# B&R Automation Studio project A2019059_Linka_Power_CP (part 4)

### Hardware.hwl.2.mine
```
BR.AS.HardwareTopology (Version=0.0.0.1)
  TimeStamps:
    TimeStamp (LogicalPath=Config1.Hardware.hw, LastWriteTime=07/08/2020 07:45:30)
  Modules:
    Module PC1 (Type=5PC910.SX02-00, X=2263, Y=-320)
    Module 5AC901.IUPS-01 (Type=5AC901.IUPS-01, X=2322, Y=-217)
    Module 5AC901.BX02-00 (Type=5AC901.BX02-00, X=2322, Y=-287)
    Module 5ACPCI_XPNM_00 (Type=5ACPCI.XPNM-00, X=2327, Y=-245)
    Module 5LS182.6-1 (Type=5LS182.6-1, X=2327, Y=-274)
    Module 5PC900_TS17_00 (Type=5PC900.TS17-00, X=2322, Y=-310)
    Module AB1.0 (Type=6PPT50.156B-10B, X=-440, Y=-300)
    Module AB2.0 (Type=6PPT50.156B-10B, X=672, Y=-281)
    Module AB4.0 (Type=6PPT50.156B-10B, X=3220, Y=-302)
    Module 0AC808.9-1 (Type=0AC808.9-1, X=2483, Y=-229)
    Module X20BB81 (Type=X20BB81, X=-440, Y=20)
    Module X20BM33 (Type=X20BM33, X=-377, Y=20)
    Module AB1.4_20xSI (Type=X20SI9100, X=-377, Y=20)
    Module X20TB52b (Type=X20TB52, X=-364, Y=46)
    Module X20TB52a (Type=X20TB52, X=-377, Y=46)
    Module X20BM33d (Type=X20BM33, X=-351, Y=20)
    Module AB1.5_6xSO (Type=X20SO6530, X=-351, Y=20)
    Module X20TB72 (Type=X20TB72, X=-351, Y=46)
    Module X20BM11 (Type=X20BM11, X=-325, Y=20)
    Module AB1.6_16xDI (Type=X20DIF371, X=-325, Y=20)
    Module X20TB1F (Type=X20TB1F, X=-325, Y=47)
    Module X20BM11a (Type=X20BM11, X=-312, Y=20)
    Module AB1.7_16xDI (Type=X20DIF371, X=-312, Y=20)
    Module X20TB1F1 (Type=X20TB1F, X=-312, Y=47)
    Module X20BM11b (Type=X20BM11, X=-299, Y=20)
    Module AB1.8_16xDO (Type=X20DOF322, X=-299, Y=20)
    Module X20TB1F2 (Type=X20TB1F, X=-299, Y=47)
    Module X20BM11c (Type=X20BM11, X=-286, Y=20)
    Module AB1.9_16xDO (Type=X20DOF322, X=-286, Y=20)
    Module X20TB1F3 (Type=X20TB1F, X=-286, Y=47)
    Module X20BM11h (Type=X20BM11, X=-273, Y=20)
    Module AB1.10_X2X (Type=X20BT9400, X=-273, Y=20)
    Module X20TB12d (Type=X20TB12, X=-273, Y=47)
    Module AB1.3_Napajanie (Type=X20PS9400, X=-390, Y=20)
    Module X20TB12 (Type=X20TB12, X=-390, Y=47)
    Module AB1.2_Powerlink (Type=X20BC1083, X=-415, Y=20)
    Module X20BB81a (Type=X20BB81, X=720, Y=20)
    Module X20BM33a (Type=X20BM33, X=783, Y=20)
    Module AB2.4_20xSI (Type=X20SI9100, X=783, Y=20)
    Module X20TB52d (Type=X20TB52, X=796, Y=46)
    Module X20TB52c (Type=X20TB52, X=783, Y=46)
    Module X20BM33e (Type=X20BM33, X=809, Y=20)
    Module AB2.5_6xSO (Type=X20SO6530, X=809, Y=20)
    Module X20TB72a (Type=X20TB72, X=809, Y=46)
    Module X20BM33h (Type=X20BM33, X=835, Y=20)
    Module AB2.6_6xSO (Type=X20SO6530, X=835, Y=20)
    Module X20TB72d (Type=X20TB72, X=835, Y=46)
    Module X20BM11d (Type=X20BM11, X=861, Y=20)
    Module AB2.7_16xDI (Type=X20DIF371, X=861, Y=20)
    Module X20TB1F4 (Type=X20TB1F, X=861, Y=47)
    Module X20BM11e (Type=X20BM11, X=874, Y=20)
    Module AB2.8_16xDI (Type=X20DIF371, X=874, Y=20)
    Module X20TB1F5 (Type=X20TB1F, X=874, Y=47)
    Module X20BM11l (Type=X20BM11, X=887, Y=20)
    Module AB2.9_16xDO (Type=X20DOF322, X=887, Y=20)
    Module X20TB1F8 (Type=X20TB1F, X=887, Y=47)
    Module X20BM11m (Type=X20BM11, X=900, Y=20)
    Module AB2.10_16xDO (Type=X20DOF322, X=900, Y=20)
    Module X20TB1F9 (Type=X20TB1F, X=900, Y=47)
    Module X20BM11i (Type=X20BM11, X=913, Y=20)
    Module AB2.11_X2X (Type=X20BT9400, X=913, Y=20)
    Module X20TB12e (Type=X20TB12, X=913, Y=47)
    Module AB2.3_Napajanie (Type=X20PS9400, X=770, Y=20)
    Module X20TB12a (Type=X20TB12, X=770, Y=47)
    Module AB2.2_Powerlink (Type=X20BC1083, X=745, Y=20)
    Module X20BB81b (Type=X20BB81, X=2019, Y=20)
    Module X20BM11f (Type=X20BM11, X=2082, Y=20)
    Module AB3.7_16xDI (Type=X20DIF371, X=2082, Y=20)
    Module X20TB1F6 (Type=X20TB1F, X=2082, Y=47)
    Module X20BM11g (Type=X20BM11, X=2095, Y=20)
    Module AB3.8_16xDO (Type=X20DOF322, X=2095, Y=20)
    Module X20TB1F7 (Type=X20TB1F, X=2095, Y=47)
    Module X20BM33b (Type=X20BM33, X=2108, Y=20)
    Module AB3.5_20xSI (Type=X20SI9100, X=2108, Y=20)
    Module X20TB52f (Type=X20TB52, X=2121, Y=46)
    Module X20TB52e (Type=X20TB52, X=2108, Y=46)
    Module X20BM33f (Type=X20BM33, X=2134, Y=20)
    Module AB3.6_6xSO (Type=X20SO6530, X=2134, Y=20)
    Module X20TB72b (Type=X20TB72, X=2134, Y=46)
    Module X20BM11j (Type=X20BM11, X=2160, Y=20)
    Module AB3.9_X2X (Type=X20BT9400, X=2160, Y=20)
    Module X20TB12f (Type=X20TB12, X=2160, Y=47)
    Module AB3.3_Napajanie (Type=X20PS9400, X=2069, Y=20)
    Module X20TB12b (Type=X20TB12, X=2069, Y=47)
    Module AB3.2_Powerlink (Type=X20BC1083, X=2044, Y=20)
    Module X20BB81c (Type=X20BB81, X=3240, Y=-2)
    Module X20BM33c (Type=X20BM33, X=3303, Y=-2)
    Module SI4.0 (Type=X20SI9100, X=3303, Y=-2)
    Module X20TB52h (Type=X20TB52, X=3316, Y=24)
    Module X20TB52g (Type=X20TB52, X=3303, Y=24)
    Module X20BM33g (Type=X20BM33, X=3329, Y=-2)
    Module SO4.0 (Type=X20SO6530, X=3329, Y=-2)
    Module X20TB72c (Type=X20TB72, X=3329, Y=24)
    Module X20BM11k (Type=X20BM11, X=3355, Y=-2)
    Module BT4.0 (Type=X20BT9400, X=3355, Y=-2)
    Module X20TB12g (Type=X20TB12, X=3355, Y=25)
    Module PS4.0 (Type=X20PS9400, X=3290, Y=-2)
    Module X20TB12c (Type=X20TB12, X=3290, Y=25)
    Module BC4.0 (Type=X20BC1083, X=3265, Y=-2)
    Module SL1_SafetyMaster (Type=X20SL8100, X=2283, Y=20)
    Module X20TB52 (Type=X20TB52, X=2330, Y=47)
    Module X20MK0211 (Type=X20MK0211, X=2286, Y=90)
    Module DM4.0 (Type=X67DM1321.L12, X=3210, Y=523)
    Module DM3.1 (Type=X67DM1321.L12, X=2090, Y=525)
    Module DM2.1_16DI/DO (Type=X67DM1321.L12, X=1024, Y=525)
    Module DM1.1_16DI/DO (Type=X67DM1321.L12, X=-282, Y=525)
    Module SI1.1 (Type=X67SI8103, X=-364, Y=525)
    Module SI1.2 (Type=X67SI8103, X=146, Y=525)
    Module SI2.1 (Type=X67SI8103, X=815, Y=525)
    Module SI2.2 (Type=X67SI8103, X=881, Y=525)
    Module SI3.1 (Type=X67SI8103, X=2005, Y=525)
    Module SI4.1 (Type=X67SI8103, X=3435, Y=523)
    Module SI4.2 (Type=X67SI8103, X=3510, Y=523)
    Module PS1.1 (Type=X67PS1300, X=-434, Y=1049)
    Module PS2.1 (Type=X67PS1300, X=1104, Y=525)
    Module PS3.1 (Type=X67PS1300, X=2467, Y=525)
    Module PS4.1 (Type=X67PS1300, X=3585, Y=523)
    Module DI2.1_8DI (Type=X67DI1371, X=785, Y=1049)
    Module X67DI1371a (Type=X67DI1371, X=3285, Y=523)
    Module DI2.2_16DI (Type=X67DI1371.L08, X=1302, Y=525)
    Module DI2.3_16DI (Type=X67DI1371.L08, X=692, Y=1049)
    Module DI2.4_16DI (Type=X67DI1371.L08, X=951, Y=525)
    Module DI2.5_16DI (Type=X67DI1371.L08, X=676, Y=525)
    Module DI1.2_16DI (Type=X67DI1371.L08, X=-185, Y=525)
    Module DI1.1_16DI (Type=X67DI1371.L08, X=36, Y=525)
    Module DI3.3_16DI (Type=X67DI1371.L08, X=2377, Y=525)
    Module DI3.2_16DI (Type=X67DI1371.L08, X=2177, Y=525)
    Module DI3.1_16DI (Type=X67DI1371.L08, X=2068, Y=1027)
    Module DS3_1 (Type=X67DS438A, X=2560, Y=525)
    Module DS3_2 (Type=X67DS438A, X=2276, Y=525)
    Module DS3_3 (Type=X67DS438A, X=2367, Y=1027)
    Module DS4_1 (Type=X67DS438A, X=3679, Y=523)
    Module DS4_2 (Type=X67DS438A, X=3795, Y=523)
    Module 0AC808.9-1a (Type=0AC808.9-1, X=2068, Y=-213)
    Module M1.0.0 (Type=8LVA23.B8015S200-0, X=-381, Y=361)
    Module M1.1.0 (Type=8LVA23.B9015S200-0, X=-171, Y=361)
    Module M1.1.1 (Type=8LVA23.B9015S200-0, X=-87, Y=365)
    Module FM4_ZdvihVytahu (Type=8EI4X5MWS10.xxxx-1, X=-442, Y=241)
    Module FM5_ManipulatorSrobovacky (Type=8EI4X5MWD10.xxxx-1, X=-229, Y=183)
    Module FM14_ManipSrobovacky (Type=8EI4X5MWS10.xxxx-1, X=2058, Y=225)
    Module SD4.0 (Type=8EI4X5MWS10.xxxx-1, X=3229, Y=259)
    Module SD4.1 (Type=8EI4X5MWS10.xxxx-1, X=3389, Y=259)
    Module M37_ManipSrobovackyOsY (Type=8LVA23.B9015S200-0, X=2118, Y=345)
    Module M4.0.0 (Type=8LVA23.B9015S200-0, X=3289, Y=379)
    Module M4.1.0 (Type=8LVA23.B8015S200-0, X=3450, Y=379)
    Module 0AC808.9-1b (Type=0AC808.9-1, X=20, Y=-221)
    Module 0AC808.9-1c (Type=0AC808.9-1, X=1139, Y=-221)
    Module 0AC808.9-1d (Type=0AC808.9-1, X=3711, Y=-203)
    Module R1_IRB120 (Type=FBD.Hilscher.PNIOGenDevDTM2.ENERGY V1.4, X=12, Y=36)
    Module R2_IRB1200 (Type=FBD.Hilscher.PNIOGenDevDTM2.ENERGY V1.4, X=1457, Y=507)
    Module X67DI1371.L08j (Type=X67DI1371.L08, X=3360, Y=523)
    Module FM5_ManipSrobovacky_ZdvihZvarania (Type=8EI4X5MWT10.xxxx-1, X=716, Y=180)
    Module M6_ZdvihZvaracky (Type=8LVA23.B9015S200-0, X=908, Y=379)
    Module M10_ManipSrobovackyOsX (Type=8LVA23.B9015S200-0, X=768, Y=380)
    Module M9_ManipSrobovackyOsY (Type=8LVA23.B9015S200-0, X=838, Y=379)
    Module FM6_ZdvihZakladacaTesnenia (Type=8EI8X8HWS10.xxxx-1, X=1024, Y=162)
    Module M4_ZdvihZakladacaTesnenia (Type=8LSA46.DB030S200-3, X=1084, Y=379)
    Module M5_PojazdZakladacaTesnenia (Type=8LSAA2.D9045S000-3, X=1265, Y=379)
    Module DS2_1 (Type=X67DS438A, X=1191, Y=525)
    Module DS2_2 (Type=X67DS438A, X=745, Y=525)
    Module DS2_3 (Type=X67DS438A, X=898, Y=1049)
    Module ModulRobot_BN2 (Type=FBD.IOLink.GenericDeviceDTM.DTMCore.BNI IOL-309-000-K024 IODD1.0.1, X=1154, Y=780)
    Module ZakladacTesnenia_BannerPotvrdeniaObsluhy_SB7 (Type=FBD.IOLink.GenericDeviceDTM.DTMCore.K50 Pro Device IODD1.1, X=1157, Y=695)
    Module SkrutkovacMatic_VysunutieHrotuSkrutkovacky_IOS7 (Type=FBD.IOLink.GenericDeviceDTM.DTMCore.Magnetic Cylinder Sensors IODD1.1, X=1157, Y=858)
    Module SkrutkovackaM6_VysunutieHrotuSkrutkovacky_IOS3 (Type=FBD.IOLink.GenericDeviceDTM.DTMCore.Magnetic Cylinder Sensors IODD1.1, X=888, Y=1324)
    Module SkrutkovackaM4_VysunutieHrotuSkrutkovacky_IOS4 (Type=FBD.IOLink.GenericDeviceDTM.DTMCore.Magnetic Cylinder Sensors IODD1.1, X=888, Y=1233)
    Module SkrutkovackaM5_VysunutieHrotuSkrutkovacky_IOS5 (Type=FBD.IOLink.GenericDeviceDTM.DTMCore.Magnetic Cylinder Sensors IODD1.1, X=888, Y=1418)
    Module Griper4F_5F_5H_SnimacOtvoreniaZatvoreniaGripra (Type=FBD.IOLink.GenericDeviceDTM.DTMCore.MMS xx-IOL-Mxx IODD1.1, X=1157, Y=931)
    Module VentilovyTerminal_VT1 (Type=FBE.FFFF0007_EX260-SPL1, X=1049, Y=0)
    Module VentilovyTerminal_VT2 (Type=FBE.FFFF0007_EX260-SPL1, X=1157, Y=0)
    Module VentilovyTerminal_VT3 (Type=FBE.FFFF0007_EX260-SPL1, X=1265, Y=0)
    Module FM7_PojazdZakladacaTesnenia (Type=8EI4X5MWS10.xxxx-1, X=1196, Y=162)
    Module StoperSkrutkovaniaMatic_SnimacPaletky_S7 (Type=FBD.IOLink.GenericDeviceDTM.DTMCore.BIS M-404-045-401-07-S4 IODD1.0.1, X=768, Y=695)
    Module StoperZakladaniaTesnenia_SnimacPaletky_S6 (Type=FBD.IOLink.GenericDeviceDTM.DTMCore.BIS M-404-045-401-07-S4 IODD1.0.1, X=762, Y=780)
    Module StoperZvarania_SnimacPaletky_S9 (Type=FBD.IOLink.GenericDeviceDTM.DTMCore.BIS M-404-045-401-07-S4 IODD1.0.1, X=762, Y=858)
    Module StoperSrobovania_SnimacPaletky_S8 (Type=FBD.IOLink.GenericDeviceDTM.DTMCore.BIS M-404-045-401-07-S4 IODD1.0.1, X=762, Y=931)
    Module DI1.3_8DI (Type=X67DI1371, X=-434, Y=525)
    Module DI1.4_8DI (Type=X67DI1371, X=-311, Y=1049)
    Module DS1_1 (Type=X67DS438A, X=-76, Y=525)
    Module DS1_2 (Type=X67DS438A, X=-171, Y=1049)
    Module ModulRobot_BN1 (Type=FBD.IOLink.GenericDeviceDTM.DTMCore.BNI IOL-309-000-K024 IODD1.0.1, X=-90, Y=680)
    Module Vytah_BannerPotvrdeniaObsluhy_SB11 (Type=FBD.IOLink.GenericDeviceDTM.DTMCore.K50 Pro Device IODD1.1, X=-90, Y=780)
    Module Vytah_SnimacPaletky_S19 (Type=FBD.IOLink.GenericDeviceDTM.DTMCore.BIS M-404-045-401-07-S4 IODD1.0.1, X=-90, Y=881)
    Module StoperSrobovania_SnimacPaletky_S16 (Type=FBD.IOLink.GenericDeviceDTM.DTMCore.BIS M-404-045-401-07-S4 IODD1.0.1, X=-90, Y=960)
    Module SkrutkovackaK30_VysunutieHrotu_IOS8 (Type=FBD.IOLink.GenericDeviceDTM.DTMCore.Magnetic Cylinder Sensors IODD1.1, X=-185, Y=1197)
    Module SkrutkovackaM4_VysunutieHrotu_IOS9 (Type=FBD.IOLink.GenericDeviceDTM.DTMCore.Magnetic Cylinder Sensors IODD1.1, X=-185, Y=1303)
    Module SkrutkovackaM5_VysunutieHrotu_IOS10 (Type=FBD.IOLink.GenericDeviceDTM.DTMCore.Magnetic Cylinder Sensors IODD1.1, X=-185, Y=1407)
    Module VentilovyTerminal_VT4 (Type=FBE.FFFF0007_EX260-SPL1, X=-229, Y=34)
    Module VentilovyTerminal_VT5 (Type=FBE.FFFF0007_EX260-SPL1, X=-118, Y=34)
    Module RJ5_P1_Srobovacka_K30 (Type=FBD.Hilscher.PNIOGenDevDTM2.RT, X=12, Y=227)
    Module RJ6_P1_Srobovacka_M5 (Type=FBD.Hilscher.PNIOGenDevDTM2.RT, X=12, Y=329)
    Module RJ7_P1_Srobovacka_M4 (Type=FBD.Hilscher.PNIOGenDevDTM2.RT, X=12, Y=428)
    Module DI3.4_8DI (Type=X67DI1371, X=2194, Y=1027)
    Module StoperSkrutkovania_SnimacPaletky_S22 (Type=FBD.IOLink.GenericDeviceDTM.DTMCore.BIS M-404-045-401-07-S4 IODD1.0.1, X=2547, Y=705)
    Module LeakegeTestA_SnimacPaletky_S23 (Type=FBD.IOLink.GenericDeviceDTM.DTMCore.BIS M-404-045-401-07-S4 IODD1.0.1, X=2547, Y=808)
    Module LeakegeTestB_SnimacPaletky_S24 (Type=FBD.IOLink.GenericDeviceDTM.DTMCore.BIS M-404-045-401-07-S4 IODD1.0.1, X=2547, Y=898)
    Module SnimacTlakuLeakeTestB_S27 (Type=FBD.IOLink.GenericDeviceDTM.DTMCore.BSP00PU IODD1.1, X=2276, Y=808)
    Module SnimacTlakuLeakeTestA_S26 (Type=FBD.IOLink.GenericDeviceDTM.DTMCore.BSP00PU IODD1.1, X=2276, Y=705)
    Module SkrutkovackaK40_VysunutieHrotuSkrutkovacky_IOS11 (Type=FBD.IOLink.GenericDeviceDTM.DTMCore.Magnetic Cylinder Sensors IODD1.1, X=2355, Y=1197)
    Module SkrutkovackaM5_VysunutieHrotuSkrutkovacky_IOS12 (Type=FBD.IOLink.GenericDeviceDTM.DTMCore.Magnetic Cylinder Sensors IODD1.1, X=2355, Y=1303)
    Module RJ2_P2_Srobovacka_M6 (Type=FBD.Hilscher.PNIOGenDevDTM2.RT, X=1457, Y=647)
    Module RJ4_P2_Srobovacka_M5 (Type=FBD.Hilscher.PNIOGenDevDTM2.RT, X=1457, Y=787)
    Module RJ3_P2_Srobovacka_M4 (Type=FBD.Hilscher.PNIOGenDevDTM2.RT, X=1457, Y=931)
    Module VentilovyTerminal_VT6 (Type=FBE.FFFF0007_EX260-SPL1, X=2195, Y=204)
    Module VentilovyTerminal_VT7 (Type=FBE.FFFF0007_EX260-SPL1, X=2330, Y=204)
    Module P3_Srobovacka_K40 (Type=FBD.Hilscher.PNIOGenDevDTM2.RT, X=2247, Y=428)
    Module P3_Srobovacka_M5 (Type=FBD.Hilscher.PNIOGenDevDTM2.RT, X=2393, Y=428)
    Module RJ1_P2_SrobovackaMatic_M4 (Type=FBD.Hilscher.PNIOGenDevDTM2.RT, X=1458, Y=1027)
    Module P1_CAM3 (Type=FBD.Hilscher.PNIOGenDevDTM2.weQube V1.4, X=215, Y=222)
  Links:
    Link (From=0AC808.9-1, To=5LS182.6-1, FromPort=ETH1, ToPort=IF1, IsRoutedByUser=False)
      Point (X=2509.96631, Y=-218.412842)
      Point (X=2509.96631, Y=-218.412842)
      Point (X=2509.96631, Y=-230.412842)
      Point (X=2509.96631, Y=-266)
      Point (X=2379.46631, Y=-266)
      Point (X=2369.46631, Y=-266)
      Point (X=2369.46631, Y=-266)
    Link (From=0AC808.9-1, To=SL1_SafetyMaster, FromPort=ETH2, ToPort=PLK1, IsRoutedByUser=True)
      Point (X=2522.96631, Y=-218.412842)
      Point (X=2522.96631, Y=-218.412842)
      Point (X=2522.96631, Y=-230.412842)
      Point (X=2522.96631, Y=-250.535934)
      Point (X=2451.52344, Y=-250.535934)
      Point (X=2451.52344, Y=131.739014)
      Point (X=2305.96631, Y=131.739014)
      Point (X=2305.96631, Y=121)
      Point (X=2305.96631, Y=94)
      Point (X=2320.96631, Y=94)
    Link (From=0AC808.9-1, To=AB1.2_Powerlink, FromPort=ETH5, ToPort=PLK1, IsRoutedByUser=True)
      Point (X=2509, Y=-205)
      Point (X=2509, Y=-205)
      Point (X=2482, Y=-205)
      Point (X=2475, Y=-205)
      Point (X=2475, Y=142)
      Point (X=-409.25, Y=142)
      Point (X=-409.25, Y=121)
      Point (X=-409.25, Y=95)
      Point (X=-401, Y=95)
    Link (From=0AC808.9-1, To=AB2.2_Powerlink, FromPort=ETH6, ToPort=PLK1, IsRoutedByUser=True)
      Point (X=2522, Y=-205)
      Point (X=2522, Y=-205)
      Point (X=2522, Y=-185)
      Point (X=2522, Y=135)
      Point (X=743.75, Y=135)
      Point (X=743.75, Y=121)
      Point (X=750.75, Y=121)
      Point (X=750.75, Y=95)
      Point (X=759, Y=95)
    Link (From=0AC808.9-1, To=AB3.2_Powerlink, FromPort=ETH7, ToPort=PLK1, IsRoutedByUser=True)
      Point (X=2062.96631, Y=95.00003)
      Point (X=2054.71631, Y=95.00003)
      Point (X=2054.71631, Y=121.000031)
      Point (X=2054.71631, Y=125)
      Point (X=2015.21179, Y=125)
      Point (X=2015.21179, Y=-3.42771578)
      Point (X=2536.00928, Y=-3.42771578)
      Point (X=2536.00928, Y=-172)
      Point (X=2535.96631, Y=-172)
      Point (X=2535.96631, Y=-185.412842)
      Point (X=2535.96631, Y=-205.412842)
      Point (X=2535.96631, Y=-205.412842)
    Link (From=0AC808.9-1, To=BC4.0, FromPort=ETH8, ToPort=PLK1, IsRoutedByUser=True)
      Point (X=2548, Y=-205)
      Point (X=2548, Y=-205)
      Point (X=2548, Y=-185)
      Point (X=2548, Y=105)
      Point (X=3271.74536, Y=105)
      Point (X=3271.74536, Y=98)
      Point (X=3271.74536, Y=73)
      Point (X=3279.99536, Y=73)
    Link (From=0AC808.9-1a, To=PC1, FromPort=ETH1, ToPort=IF3, IsRoutedByUser=False)
      Point (X=2094.96631, Y=-202)
      Point (X=2094.96631, Y=-202)
      Point (X=2094.96631, Y=-214)
      Point (X=2094.96631, Y=-225)
      Point (X=2188.96631, Y=-225)
      Point (X=2188.96631, Y=-115)
      Point (X=2273.46631, Y=-115)
      Point (X=2273.46631, Y=-122)
      Point (X=2273.46631, Y=-127)
      Point (X=2273.46631, Y=-127)
    Link (From=0AC808.9-1a, To=0AC808.9-1b, FromPort=ETH5, ToPort=ETH1, IsRoutedByUser=True)
      Point (X=2094, Y=-189)
      Point (X=2094, Y=-189)
      Point (X=2067, Y=-189)
      Point (X=1938.21008, Y=-189)
      Point (X=1938.21008, Y=-322)
      Point (X=46, Y=-322)
      Point (X=46, Y=-222)
      Point (X=46, Y=-210)
      Point (X=46, Y=-210)
    Link (From=0AC808.9-1a, To=0AC808.9-1c, FromPort=ETH6, ToPort=ETH1, IsRoutedByUser=True)
      Point (X=2107, Y=-189)
      Point (X=2107, Y=-189)
      Point (X=2107, Y=-169)
      Point (X=2107, Y=-149.293823)
      Point (X=1841.18677, Y=-149.293823)
      Point (X=1841.18677, Y=-235)
      Point (X=1165, Y=-235)
      Point (X=1165, Y=-222)
      Point (X=1165, Y=-210)
      Point (X=1165, Y=-210)
    Link (From=0AC808.9-1a, To=0AC808.9-1d, FromPort=ETH8, ToPort=ETH8, IsRoutedByUser=True)
      Point (X=2133, Y=-189)
      Point (X=2133, Y=-189)
      Point (X=2133, Y=-169)
      Point (X=2133, Y=-48.8859749)
      Point (X=3776.99536, Y=-48.8859749)
      Point (X=3776.99536, Y=-159)
      Point (X=3776.99536, Y=-179)
      Point (X=3776.99536, Y=-179)
    Link (From=0AC808.9-1b, To=AB1.0, FromPort=ETH5, ToPort=ETH1, IsRoutedByUser=True)
      Point (X=-295.1, Y=-114.7)
      Point (X=-295.1, Y=-114.7)
      Point (X=-295.1, Y=-109.7)
      Point (X=-295.1, Y=-105)
      Point (X=-17.4831429, Y=-105)
      Point (X=-17.4831429, Y=-197.130936)
      Point (X=19.1028137, Y=-197.130936)
      Point (X=46.1028137, Y=-197.130936)
      Point (X=46.1028137, Y=-197.130936)
    Link (From=0AC808.9-1c, To=AB2.0, FromPort=ETH5, ToPort=ETH1, IsRoutedByUser=True)
      Point (X=1165, Y=-197)
      Point (X=1165, Y=-197)
      Point (X=1138, Y=-197)
      Point (X=1131, Y=-197)
      Point (X=1131, Y=-85)
      Point (X=817.7252, Y=-85)
      Point (X=817.7252, Y=-91.13939)
      Point (X=817.7252, Y=-96.13939)
      Point (X=817.7252, Y=-96.13939)
    Link (From=0AC808.9-1d, To=AB4.0, FromPort=ETH5, ToPort=ETH1, IsRoutedByUser=True)
      Point (X=3366.86157, Y=-116.7)
      Point (X=3366.86157, Y=-116.7)
      Point (X=3366.86157, Y=-111.7)
      Point (X=3366.86157, Y=-103.758408)
      Point (X=3677.95923, Y=-103.758408)
      Point (X=3677.95923, Y=-179.028076)
      Point (X=3712.47632, Y=-179.028076)
      Point (X=3739.47632, Y=-179.028076)
      Point (X=3739.47632, Y=-179.028076)
    Link (From=5ACPCI_XPNM_00, To=R1_IRB120, FromPort=IF1, ToPort=PN1, IsRoutedByUser=True)
      Point (X=2368, Y=-237)
      Point (X=2368, Y=-237)
      Point (X=2378, Y=-237)
      Point (X=2385, Y=-237)
      Point (X=2385, Y=-78)
      Point (X=315, Y=-78)
      Point (X=315, Y=95)
      Point (X=31, Y=95)
      Point (X=31, Y=87)
      Point (X=31, Y=75)
      Point (X=31, Y=75)
    Link (From=AB1.10_X2X, To=DI1.3_8DI, FromPort=X2X1, ToPort=X2X1, IsRoutedByUser=False)
      Point (X=-424, Y=537)
      Point (X=-424, Y=537)
      Point (X=-424, Y=524)
      Point (X=-424, Y=515)
      Point (X=-455, Y=515)
      Point (X=-455, Y=175)
      Point (X=-245, Y=175)
      Point (X=-245, Y=64)
      Point (X=-259, Y=64)
      Point (X=-266, Y=64)
      Point (X=-266, Y=64)
    Link (From=AB1.2_Powerlink, To=FM4_ZdvihVytahu, FromPort=PLK2, ToPort=PLK1, IsRoutedByUser=False)
      Point (X=-434.3, Y=251.5)
      Point (X=-434.3, Y=251.5)
      Point (X=-434.3, Y=240.5)
      Point (X=-434.3, Y=235)
      Point (X=-401, Y=235)
      Point (X=-401, Y=121)
      Point (X=-401, Y=110)
      Point (X=-401, Y=110)
    Link (From=AB2.11_X2X, To=DI2.5_16DI, FromPort=X2X1, ToPort=X2X1, IsRoutedByUser=False)
      Point (X=686, Y=537)
      Point (X=686, Y=537)
      Point (X=686, Y=524)
      Point (X=686, Y=15)
      Point (X=941, Y=15)
      Point (X=941, Y=64)
      Point (X=927, Y=64)
      Point (X=920, Y=64)
      Point (X=920, Y=64)
    Link (From=AB2.2_Powerlink, To=FM5_ManipSrobovacky_ZdvihZvarania, FromPort=PLK2, ToPort=PLK1, IsRoutedByUser=False)
      Point (X=723.699951, Y=190.5)
      Point (X=723.699951, Y=190.5)
      Point (X=723.699951, Y=179.5)
      Point (X=723.699951, Y=175)
      Point (X=755, Y=175)
      Point (X=755, Y=121)
      Point (X=755, Y=110)
      Point (X=755, Y=110)
    Link (From=AB3.2_Powerlink, To=FM14_ManipSrobovacky, FromPort=PLK2, ToPort=PLK1, IsRoutedByUser=False)
      Point (X=2066.66626, Y=235.5)
      Point (X=2066.66626, Y=235.5)
      Point (X=2066.66626, Y=224.5)
      Point (X=2066.66626, Y=215)
      Point (X=2062.96631, Y=215)
      Point (X=2062.96631, Y=121)
      Point (X=2062.96631, Y=110)
      Point (X=2062.96631, Y=110)
    Link (From=AB3.9_X2X, To=SI3.1, FromPort=X2X1, ToPort=X2X1, IsRoutedByUser=True)
      Point (X=2015.96631, Y=537)
      Point (X=2015.96631, Y=537)
      Point (X=2015.96631, Y=524)
      Point (X=2015.96631, Y=181.499237)
      Point (X=2192.713, Y=181.499237)
      Point (X=2192.713, Y=64)
      Point (X=2178.96631, Y=64)
      Point (X=2171.96631, Y=64)
      Point (X=2171.96631, Y=64)
    Link (From=BT4.0, To=DM4.0, FromPort=X2X1, ToPort=X2X1, IsRoutedByUser=True)
      Point (X=3363.96167, Y=42)
      Point (X=3363.96167, Y=42)
      Point (X=3370.96167, Y=42)
      Point (X=3376.96167, Y=42)
      Point (X=3376.96167, Y=473)
      Point (X=3221.96167, Y=473)
      Point (X=3221.96167, Y=522)
      Point (X=3221.96167, Y=535)
      Point (X=3221.96167, Y=535)
    Link (From=DI1.1_16DI, To=DS1_1, FromPort=X2X1, ToPort=X2X2, IsRoutedByUser=False)
      Point (X=-34, Y=537)
      Point (X=-34, Y=537)
      Point (X=9, Y=537)
      Point (X=35, Y=537)
      Point (X=46, Y=537)
      Point (X=46, Y=537)
    Link (From=DI1.1_16DI, To=SI1.2, FromPort=X2X2, ToPort=X2X1, IsRoutedByUser=False)
      Point (X=78, Y=537)
      Point (X=78, Y=537)
      Point (X=90, Y=537)
      Point (X=145.228729, Y=537)
      Point (X=156.228729, Y=537)
      Point (X=156.228729, Y=537)
    Link (From=DI1.2_16DI, To=DM1.1_16DI/DO, FromPort=X2X1, ToPort=X2X2, IsRoutedByUser=False)
      Point (X=-240, Y=537)
      Point (X=-240, Y=537)
      Point (X=-228, Y=537)
      Point (X=-186, Y=537)
      Point (X=-175, Y=537)
      Point (X=-175, Y=537)
    Link (From=DI1.2_16DI, To=DS1_1, FromPort=X2X2, ToPort=X2X1, IsRoutedByUser=False)
      Point (X=-143, Y=537)
      Point (X=-143, Y=537)
      Point (X=-131, Y=537)
      Point (X=-110, Y=537)
      Point (X=-66, Y=537)
      Point (X=-66, Y=537)
    Link (From=DI1.3_8DI, To=SI1.1, FromPort=X2X2, ToPort=X2X1, IsRoutedByUser=False)
      Point (X=-392, Y=537)
      Point (X=-392, Y=537)
      Point (X=-380, Y=537)
      Point (X=-365, Y=537)
      Point (X=-354, Y=537)
      Point (X=-354, Y=537)
    Link (From=DI1.4_8DI, To=PS1.1, FromPort=X2X1, ToPort=X2X2, IsRoutedByUser=False)
      Point (X=-392, Y=1061)
      Point (X=-392, Y=1061)
      Point (X=-380, Y=1061)
      Point (X=-312, Y=1061)
      Point (X=-301, Y=1061)
      Point (X=-301, Y=1061)
    Link (From=DI1.4_8DI, To=DS1_2, FromPort=X2X2, ToPort=X2X1, IsRoutedByUser=False)
      Point (X=-269, Y=1061)
      Point (X=-269, Y=1061)
      Point (X=-257, Y=1061)
      Point (X=-205, Y=1061)
      Point (X=-161, Y=1061)
      Point (X=-161, Y=1061)
    Link (From=DI2.1_8DI, To=DI2.3_16DI, FromPort=X2X1, ToPort=X2X2, IsRoutedByUser=False)
      Point (X=734.020569, Y=1061.34363)
      Point (X=734.020569, Y=1061.34363)
      Point (X=746.020569, Y=1061.34363)
      Point (X=784, Y=1061.34363)
      Point (X=795, Y=1061.34363)
      Point (X=795, Y=1061.34363)
    Link (From=DI2.1_8DI, To=DS2_3, FromPort=X2X2, ToPort=X2X1, IsRoutedByUser=False)
      Point (X=827, Y=1061.34363)
      Point (X=827, Y=1061.34363)
      Point (X=839, Y=1061.34363)
      Point (X=864.4114, Y=1061.34363)
      Point (X=908.4114, Y=1061.34363)
      Point (X=908.4114, Y=1061.34363)
    Link (From=DI2.2_16DI, To=DS2_1, FromPort=X2X1, ToPort=X2X2, IsRoutedByUser=False)
      Point (X=1233, Y=537)
      Point (X=1233, Y=537)
      Point (X=1276, Y=537)
      Point (X=1301, Y=537)
      Point (X=1312, Y=537)
      Point (X=1312, Y=537)
    Link (From=DI2.2_16DI, To=DI2.3_16DI, FromPort=X2X2, ToPort=X2X1, IsRoutedByUser=True)
      Point (X=1344, Y=537)
      Point (X=1344, Y=537)
      Point (X=1356, Y=537)
      Point (X=1361, Y=537)
      Point (X=1361, Y=705)
      Point (X=1361.66431, Y=705)
      Point (X=1361.66431, Y=1023.05377)
      Point (X=681, Y=1023.05377)
      Point (X=681, Y=1061)
      Point (X=691, Y=1061)
      Point (X=702, Y=1061)
      Point (X=702, Y=1061)
    Link (From=DI2.4_16DI, To=SI2.2, FromPort=X2X1, ToPort=X2X2, IsRoutedByUser=False)
      Point (X=923, Y=537)
      Point (X=923, Y=537)
      Point (X=935, Y=537)
      Point (X=950.4114, Y=537)
      Point (X=961.4114, Y=537)
      Point (X=961.4114, Y=537)
    Link (From=DI2.4_16DI, To=DM2.1_16DI/DO, FromPort=X2X2, ToPort=X2X1, IsRoutedByUser=False)
      Point (X=993.4114, Y=537)
      Point (X=993.4114, Y=537)
      Point (X=1005.41138, Y=537)
      Point (X=1023, Y=537)
      Point (X=1034, Y=537)
      Point (X=1034, Y=537)
    Link (From=DI2.5_16DI, To=DS2_2, FromPort=X2X2, ToPort=X2X1, IsRoutedByUser=True)
      Point (X=718, Y=537)
      Point (X=718, Y=537)
      Point (X=730, Y=537)
      Point (X=739.2722, Y=537)
      Point (X=711.020569, Y=537)
      Point (X=755.020569, Y=537)
      Point (X=755.020569, Y=537)
    Link (From=DI3.1_16DI, To=DS3_1, FromPort=X2X1, ToPort=X2X2, IsRoutedByUser=True)
      Point (X=2079.41528, Y=1039)
      Point (X=2079.41528, Y=1039)
      Point (X=2068.41528, Y=1039)
      Point (X=2001.96631, Y=1039)
      Point (X=2001.96631, Y=996.794067)
      Point (X=2655.96631, Y=996.794067)
      Point (X=2655.96631, Y=537)
      Point (X=2645.96631, Y=537)
      Point (X=2602.96631, Y=537)
      Point (X=2602.96631, Y=537)
    Link (From=DI3.1_16DI, To=DI3.4_8DI, FromPort=X2X2, ToPort=X2X1, IsRoutedByUser=False)
      Point (X=2110, Y=1039)
      Point (X=2110, Y=1039)
      Point (X=2122, Y=1039)
      Point (X=2193, Y=1039)
      Point (X=2204, Y=1039)
      Point (X=2204, Y=1039)
    Link (From=DI3.2_16DI, To=DM3.1, FromPort=X2X1, ToPort=X2X2, IsRoutedByUser=False)
      Point (X=2132.96631, Y=537)
      Point (X=2132.96631, Y=537)
      Point (X=2144.96631, Y=537)
      Point (X=2176.96631, Y=537)
      Point (X=2187.96631, Y=537)
      Point (X=2187.96631, Y=537)
    Link (From=DI3.2_16DI, To=DS3_2, FromPort=X2X2, ToPort=X2X1, IsRoutedByUser=False)
      Point (X=2219.96631, Y=537)
      Point (X=2219.96631, Y=537)
      Point (X=2231.96631, Y=537)
      Point (X=2243.46631, Y=537)
      Point (X=2287.46631, Y=537)
      Point (X=2287.46631, Y=537)
    Link (From=DI3.3_16DI, To=DS3_2, FromPort=X2X1, ToPort=X2X2, IsRoutedByUser=False)
      Point (X=2319.46631, Y=537)
      Point (X=2319.46631, Y=537)
      Point (X=2362.46631, Y=537)
      Point (X=2376.96631, Y=537)
      Point (X=2387.96631, Y=537)
      Point (X=2387.96631, Y=537)
    Link (From=DI3.3_16DI, To=PS3.1, FromPort=X2X2, ToPort=X2X1, IsRoutedByUser=False)
      Point (X=2419.96631, Y=537)
      Point (X=2419.96631, Y=537)
      Point (X=2431.96631, Y=537)
      Point (X=2466.96631, Y=537)
      Point (X=2477.96631, Y=537)
      Point (X=2477.96631, Y=537)
    Link (From=DI3.4_8DI, To=DS3_3, FromPort=X2X2, ToPort=X2X1, IsRoutedByUser=False)
      Point (X=2237.644, Y=1039)
      Point (X=2237.644, Y=1039)
      Point (X=2249.644, Y=1039)
      Point (X=2333.96631, Y=1039)
      Point (X=2377.96631, Y=1039)
      Point (X=2377.96631, Y=1039)
    Link (From=DM1.1_16DI/DO, To=SI1.1, FromPort=X2X1, ToPort=X2X2, IsRoutedByUser=False)
      Point (X=-322, Y=537)
      Point (X=-322, Y=537)
      Point (X=-310, Y=537)
      Point (X=-283, Y=537)
      Point (X=-272, Y=537)
      Point (X=-272, Y=537)
    Link (From=DM2.1_16DI/DO, To=PS2.1, FromPort=X2X2, ToPort=X2X1, IsRoutedByUser=False)
      Point (X=1066, Y=537)
      Point (X=1066, Y=537)
      Point (X=1078, Y=537)
      Point (X=1103, Y=537)
      Point (X=1114, Y=537)
      Point (X=1114, Y=537)
    Link (From=DM3.1, To=SI3.1, FromPort=X2X1, ToPort=X2X2, IsRoutedByUser=False)
      Point (X=2047.96631, Y=537)
      Point (X=2047.96631, Y=537)
      Point (X=2059.96631, Y=537)
      Point (X=2089.96631, Y=537)
      Point (X=2100.96631, Y=537)
      Point (X=2100.96631, Y=537)
    Link (From=DM4.0, To=X67DI1371a, FromPort=X2X2, ToPort=X2X1, IsRoutedByUser=False)
      Point (X=3253.96167, Y=535)
      Point (X=3253.96167, Y=535)
      Point (X=3265.96167, Y=535)
      Point (X=3285.96167, Y=535)
      Point (X=3296.96167, Y=535)
      Point (X=3296.96167, Y=535)
    Link (From=DS1_1, To=ModulRobot_BN1, FromPort=IF1, ToPort=IO-Link1, IsRoutedByUser=False)
      Point (X=-71, Y=719)
      Point (X=-71, Y=719)
      Point (X=-71, Y=731)
      Point (X=-71, Y=745)
      Point (X=-95, Y=745)
      Point (X=-95, Y=675)
      Point (X=-73.5, Y=675)
      Point (X=-73.5, Y=611)
      Point (X=-73.5, Y=560)
      Point (X=-66, Y=560)
    Link (From=DS1_1, To=Vytah_BannerPotvrdeniaObsluhy_SB11, FromPort=IF2, ToPort=IO-Link1, IsRoutedByUser=False)
      Point (X=-71, Y=819)
      Point (X=-71, Y=819)
      Point (X=-71, Y=831)
      Point (X=-71, Y=845)
      Point (X=-102, Y=845)
      Point (X=-102, Y=668)
      Point (X=-66, Y=668)
      Point (X=-66, Y=611)
      Point (X=-66, Y=584)
      Point (X=-66, Y=584)
    Link (From=DS1_1, To=Vytah_SnimacPaletky_S19, FromPort=IF3, ToPort=IO-Link1, IsRoutedByUser=False)
      Point (X=-71, Y=920)
      Point (X=-71, Y=920)
      Point (X=-71, Y=932)
      Point (X=-71, Y=945)
      Point (X=-109, Y=945)
      Point (X=-109, Y=661)
      Point (X=-42.25, Y=661)
      Point (X=-42.25, Y=611)
      Point (X=-42.25, Y=560)
      Point (X=-34, Y=560)
    Link (From=DS1_1, To=StoperSrobovania_SnimacPaletky_S16, FromPort=IF4, ToPort=IO-Link1, IsRoutedByUser=False)
      Point (X=-71, Y=999.794067)
      Point (X=-71, Y=999.794067)
      Point (X=-71, Y=1011.79407)
      Point (X=-71, Y=1025)
      Point (X=-116, Y=1025)
      Point (X=-116, Y=654)
      Point (X=-34, Y=654)
      Point (X=-34, Y=611)
      Point (X=-34, Y=584)
      Point (X=-34, Y=584)
    Link (From=DS1_2, To=SkrutkovackaK30_VysunutieHrotu_IOS8, FromPort=IF1, ToPort=IO-Link1, IsRoutedByUser=False)
      Point (X=-166, Y=1236.79407)
      Point (X=-166, Y=1236.79407)
      Point (X=-166, Y=1248.79407)
      Point (X=-166, Y=1255)
      Point (X=-195, Y=1255)
      Point (X=-195, Y=1185)
      Point (X=-168.5, Y=1185)
      Point (X=-168.5, Y=1135)
      Point (X=-168.5, Y=1084)
      Point (X=-161, Y=1084)
    Link (From=DS1_2, To=SkrutkovackaM4_VysunutieHrotu_IOS9, FromPort=IF2, ToPort=IO-Link1, IsRoutedByUser=False)
      Point (X=-166, Y=1342.79407)
      Point (X=-166, Y=1342.79407)
      Point (X=-166, Y=1354.79407)
      Point (X=-166, Y=1365)
      Point (X=-202, Y=1365)
      Point (X=-202, Y=1178)
      Point (X=-161, Y=1178)
      Point (X=-161, Y=1135)
      Point (X=-161, Y=1108)
      Point (X=-161, Y=1108)
    Link (From=DS1_2, To=SkrutkovackaM5_VysunutieHrotu_IOS10, FromPort=IF3, ToPort=IO-Link1, IsRoutedByUser=False)
      Point (X=-166, Y=1446.79407)
      Point (X=-166, Y=1446.79407)
      Point (X=-166, Y=1458.79407)
      Point (X=-166, Y=1465)
      Point (X=-209, Y=1465)
      Point (X=-209, Y=1171)
      Point (X=-137.25, Y=1171)
      Point (X=-137.25, Y=1135)
      Point (X=-137.25, Y=1084)
      Point (X=-129, Y=1084)
    Link (From=DS2_1, To=PS2.1, FromPort=X2X1, ToPort=X2X2, IsRoutedByUser=True)
      Point (X=1146, Y=537)
      Point (X=1146, Y=537)
      Point (X=1158, Y=537)
      Point (X=1157, Y=537)
      Point (X=1201, Y=537)
      Point (X=1201, Y=537)
    Link (From=DS2_1, To=ModulRobot_BN2, FromPort=IF1, ToPort=IO-Link1, IsRoutedByUser=True)
      Point (X=1173, Y=819)
      Point (X=1173, Y=819)
      Point (X=1173, Y=831)
      Point (X=1173, Y=845)
      Point (X=1141, Y=845)
      Point (X=1141, Y=640.4898)
      Point (X=1193.5, Y=640.4898)
      Point (X=1193.5, Y=611)
      Point (X=1193.5, Y=560)
      Point (X=1201, Y=560)
    Link (From=DS2_1, To=ZakladacTesnenia_BannerPotvrdeniaObsluhy_SB7, FromPort=IF2, ToPort=IO-Link1, IsRoutedByUser=True)
      Point (X=1176, Y=734)
      Point (X=1176, Y=734)
      Point (X=1176, Y=746)
      Point (X=1176, Y=757.0421)
      Point (X=1148.20361, Y=757.0421)
      Point (X=1148.20361, Y=671)
      Point (X=1201, Y=671)
      Point (X=1201, Y=611)
      Point (X=1201, Y=584)
      Point (X=1201, Y=584)
    Link (From=DS2_1, To=SkrutkovacMatic_VysunutieHrotuSkrutkovacky_IOS7, FromPort=IF3, ToPort=IO-Link1, IsRoutedByUser=True)
      Point (X=1176, Y=897.6584)
      Point (X=1176, Y=897.6584)
      Point (X=1176, Y=909.6584)
      Point (X=1176, Y=922.5661)
      Point (X=1265.73535, Y=922.5661)
      Point (X=1265.73535, Y=678)
      Point (X=1224.75, Y=678)
      Point (X=1224.75, Y=611)
      Point (X=1224.75, Y=560)
      Point (X=1233, Y=560)
    Link (From=DS2_1, To=Griper4F_5F_5H_SnimacOtvoreniaZatvoreniaGripra, FromPort=IF4, ToPort=IO-Link1, IsRoutedByUser=True)
      Point (X=1176, Y=970.136353)
      Point (X=1176, Y=970.136353)
      Point (X=1176, Y=982.136353)
      Point (X=1176, Y=990.2379)
      Point (X=1285.324, Y=990.2379)
      Point (X=1285.324, Y=665.0665)
      Point (X=1233, Y=665.0665)
      Point (X=1233, Y=611)
      Point (X=1233, Y=584)
      Point (X=1233, Y=584)
    Link (From=DS2_2, To=SI2.1, FromPort=X2X2, ToPort=X2X1, IsRoutedByUser=False)
      Point (X=787, Y=537)
      Point (X=787, Y=537)
      Point (X=830, Y=537)
      Point (X=862.980469, Y=537)
      Point (X=862.980469, Y=516)
      Point (X=875, Y=516)
      Point (X=875, Y=515)
      Point (X=805, Y=515)
      Point (X=805, Y=537)
      Point (X=814, Y=537)
      Point (X=825, Y=537)
      Point (X=825, Y=537)
    Link (From=DS2_2, To=StoperZakladaniaTesnenia_SnimacPaletky_S6, FromPort=IF1, ToPort=IO-Link1, IsRoutedByUser=False)
      Point (X=755, Y=560)
      Point (X=747.5, Y=560)
      Point (X=747.5, Y=611)
      Point (X=747.5, Y=845)
      Point (X=781, Y=845)
      Point (X=781, Y=831)
      Point (X=781, Y=819)
      Point (X=781, Y=819)
    Link (From=DS2_2, To=StoperSkrutkovaniaMatic_SnimacPaletky_S7, FromPort=IF2, ToPort=IO-Link1, IsRoutedByUser=False)
      Point (X=755, Y=584)
      Point (X=755, Y=584)
      Point (X=755, Y=611)
      Point (X=755, Y=755)
      Point (X=787, Y=755)
      Point (X=787, Y=746)
      Point (X=787, Y=734)
      Point (X=787, Y=734)
    Link (From=DS2_2, To=StoperSrobovania_SnimacPaletky_S8, FromPort=IF3, ToPort=IO-Link1, IsRoutedByUser=False)
      Point (X=787, Y=560)
      Point (X=778.75, Y=560)
      Point (X=778.75, Y=611)
      Point (X=778.75, Y=632)
      Point (X=751, Y=632)
      Point (X=751, Y=995)
      Point (X=781, Y=995)
      Point (X=781, Y=982)
      Point (X=781, Y=970)
      Point (X=781, Y=970)
    Link (From=DS2_2, To=StoperZvarania_SnimacPaletky_S9, FromPort=IF4, ToPort=IO-Link1, IsRoutedByUser=False)
      Point (X=787, Y=584)
      Point (X=787, Y=584)
      Point (X=787, Y=611)
      Point (X=787, Y=625)
      Point (X=737, Y=625)
      Point (X=737, Y=915)
      Point (X=781, Y=915)
      Point (X=781, Y=909)
      Point (X=781, Y=897)
      Point (X=781, Y=897)
    Link (From=DS2_3, To=SkrutkovackaM6_VysunutieHrotuSkrutkovacky_IOS3, FromPort=IF1, ToPort=IO-Link1, IsRoutedByUser=True)
      Point (X=907, Y=1363.67969)
      Point (X=907, Y=1363.67969)
      Point (X=907, Y=1375.67969)
      Point (X=907, Y=1385)
      Point (X=850.45636, Y=1385)
      Point (X=850.45636, Y=1204.68347)
      Point (X=900.9114, Y=1204.68347)
      Point (X=900.9114, Y=1135.34363)
      Point (X=900.9114, Y=1084.34363)
      Point (X=908.4114, Y=1084.34363)
    Link (From=DS2_3, To=SkrutkovackaM4_VysunutieHrotuSkrutkovacky_IOS4, FromPort=IF2, ToPort=IO-Link1, IsRoutedByUser=False)
      Point (X=907, Y=1272.05566)
      Point (X=907, Y=1272.05566)
      Point (X=907, Y=1284.05566)
      Point (X=907, Y=1295)
      Point (X=867, Y=1295)
      Point (X=867, Y=1225)
      Point (X=908.4114, Y=1225)
      Point (X=908.4114, Y=1135.34363)
      Point (X=908.4114, Y=1108.34363)
      Point (X=908.4114, Y=1108.34363)
    Link (From=DS2_3, To=SkrutkovackaM5_VysunutieHrotuSkrutkovacky_IOS5, FromPort=IF3, ToPort=IO-Link1, IsRoutedByUser=True)
      Point (X=907, Y=1457.16833)
      Point (X=907, Y=1457.16833)
      Point (X=907, Y=1469.16833)
      Point (X=907, Y=1486.75977)
      Point (X=999.329956, Y=1486.75977)
      Point (X=999.329956, Y=1218)
      Point (X=932.1614, Y=1218)
      Point (X=932.1614, Y=1135.34363)
      Point (X=932.1614, Y=1084.34363)
      Point (X=940.4114, Y=1084.34363)
    Link (From=DS3_1, To=PS3.1, FromPort=X2X1, ToPort=X2X2, IsRoutedByUser=False)
      Point (X=2509.96631, Y=537)
      Point (X=2509.96631, Y=537)
      Point (X=2521.96631, Y=537)
      Point (X=2526.96631, Y=537)
      Point (X=2570.96631, Y=537)
      Point (X=2570.96631, Y=537)
    Link (From=DS3_1, To=StoperSkrutkovania_SnimacPaletky_S22, FromPort=IF1, ToPort=IO-Link1, IsRoutedByUser=False)
      Point (X=2567.644, Y=744.451538)
      Point (X=2567.644, Y=744.451538)
      Point (X=2567.644, Y=756.451538)
      Point (X=2567.644, Y=765)
      Point (X=2538.96631, Y=765)
      Point (X=2538.96631, Y=695)
      Point (X=2563.46631, Y=695)
      Point (X=2563.46631, Y=611)
      Point (X=2563.46631, Y=560)
      Point (X=2570.96631, Y=560)
    Link (From=DS3_1, To=LeakegeTestA_SnimacPaletky_S23, FromPort=IF2, ToPort=IO-Link1, IsRoutedByUser=False)
      Point (X=2567.644, Y=847)
      Point (X=2567.644, Y=847)
      Point (X=2567.644, Y=859)
      Point (X=2567.644, Y=865)
      Point (X=2531.96631, Y=865)
      Point (X=2531.96631, Y=688)
      Point (X=2570.96631, Y=688)
      Point (X=2570.96631, Y=611)
      Point (X=2570.96631, Y=584)
      Point (X=2570.96631, Y=584)
    Link (From=DS3_1, To=LeakegeTestB_SnimacPaletky_S24, FromPort=IF3, ToPort=IO-Link1, IsRoutedByUser=False)
      Point (X=2567.644, Y=937)
      Point (X=2567.644, Y=937)
      Point (X=2567.644, Y=949)
      Point (X=2567.644, Y=955)
      Point (X=2524.96631, Y=955)
      Point (X=2524.96631, Y=681)
      Point (X=2594.71631, Y=681)
      Point (X=2594.71631, Y=611)
      Point (X=2594.71631, Y=560)
      Point (X=2602.96631, Y=560)
    Link (From=DS3_2, To=SnimacTlakuLeakeTestA_S26, FromPort=IF1, ToPort=IO-Link1, IsRoutedByUser=False)
      Point (X=2295.96631, Y=744)
      Point (X=2295.96631, Y=744)
      Point (X=2295.96631, Y=756)
      Point (X=2295.96631, Y=765)
      Point (X=2268.96631, Y=765)
      Point (X=2268.96631, Y=695)
      Point (X=2279.46631, Y=695)
      Point (X=2279.46631, Y=611)
      Point (X=2279.46631, Y=560)
      Point (X=2286.96631, Y=560)
    Link (From=DS3_2, To=SnimacTlakuLeakeTestB_S27, FromPort=IF2, ToPort=IO-Link1, IsRoutedByUser=False)
      Point (X=2295.96631, Y=847)
      Point (X=2295.96631, Y=847)
      Point (X=2295.96631, Y=859)
      Point (X=2295.96631, Y=865)
      Point (X=2261.96631, Y=865)
      Point (X=2261.96631, Y=688)
      Point (X=2286.96631, Y=688)
      Point (X=2286.96631, Y=611)
      Point (X=2286.96631, Y=584)
      Point (X=2286.96631, Y=584)
    Link (From=DS3_3, To=SkrutkovackaK40_VysunutieHrotuSkrutkovacky_IOS11, FromPort=IF1, ToPort=IO-Link1, IsRoutedByUser=False)
      Point (X=2374.96631, Y=1236)
      Point (X=2374.96631, Y=1236)
      Point (X=2374.96631, Y=1248)
      Point (X=2374.96631, Y=1255)
      Point (X=2348.96631, Y=1255)
      Point (X=2348.96631, Y=1185)
      Point (X=2370.46631, Y=1185)
      Point (X=2370.46631, Y=1113)
      Point (X=2370.46631, Y=1062)
      Point (X=2377.96631, Y=1062)
    Link (From=DS3_3, To=SkrutkovackaM5_VysunutieHrotuSkrutkovacky_IOS12, FromPort=IF2, ToPort=IO-Link1, IsRoutedByUser=False)
      Point (X=2374.96631, Y=1342)
      Point (X=2374.96631, Y=1342)
      Point (X=2374.96631, Y=1354)
      Point (X=2374.96631, Y=1365)
      Point (X=2341.96631, Y=1365)
      Point (X=2341.96631, Y=1178)
      Point (X=2377.96631, Y=1178)
      Point (X=2377.96631, Y=1113)
      Point (X=2377.96631, Y=1086)
      Point (X=2377.96631, Y=1086)
    Link (From=DS4_1, To=PS4.1, FromPort=X2X1, ToPort=X2X2, IsRoutedByUser=False)
      Point (X=3628.96167, Y=535)
      Point (X=3628.96167, Y=535)
      Point (X=3640.96167, Y=535)
      Point (X=3646.96167, Y=535)
      Point (X=3690.96167, Y=535)
      Point (X=3690.96167, Y=535)
    Link (From=DS4_1, To=DS4_2, FromPort=X2X2, ToPort=X2X1, IsRoutedByUser=False)
      Point (X=3722.96167, Y=535)
      Point (X=3722.96167, Y=535)
      Point (X=3765.96167, Y=535)
      Point (X=3762.96167, Y=535)
      Point (X=3806.96167, Y=535)
      Point (X=3806.96167, Y=535)
    Link (From=FM14_ManipSrobovacky, To=VentilovyTerminal_VT6, FromPort=PLK2, ToPort=PLK1, IsRoutedByUser=False)
      Point (X=2074.1, Y=235.5)
      Point (X=2074.1, Y=235.5)
      Point (X=2074.1, Y=224.5)
      Point (X=2074.1, Y=215)
      Point (X=2117, Y=215)
      Point (X=2117, Y=286)
      Point (X=2228.644, Y=286)
      Point (X=2228.644, Y=255)
      Point (X=2228.644, Y=248)
      Point (X=2228.644, Y=248)
    Link (From=FM14_ManipSrobovacky, To=M37_ManipSrobovackyOsY, FromPort=EC1, ToPort=EC, IsRoutedByUser=False)
      Point (X=2140.46631, Y=351.1)
      Point (X=2140.46631, Y=351.1)
      Point (X=2140.46631, Y=344.1)
      Point (X=2140.46631, Y=264)
      Point (X=2105.96631, Y=264)
      Point (X=2083.96631, Y=264)
      Point (X=2083.96631, Y=264)
    Link (From=FM14_ManipSrobovacky, To=M37_ManipSrobovackyOsY, FromPort=MT1, ToPort=MT, IsRoutedByUser=False)
      Point (X=2168.46631, Y=351.1)
      Point (X=2168.46631, Y=351.1)
      Point (X=2168.46631, Y=344.1)
      Point (X=2168.46631, Y=273.3)
      Point (X=2105.56641, Y=273.3)
      Point (X=2085.56641, Y=273.3)
      Point (X=2085.56641, Y=273.3)
    Link (From=FM4_ZdvihVytahu, To=FM5_ManipulatorSrobovacky, FromPort=PLK2, ToPort=PLK1, IsRoutedByUser=False)
      Point (X=-425.9, Y=251.5)
      Point (X=-425.9, Y=251.5)
      Point (X=-425.9, Y=240.5)
      Point (X=-425.9, Y=193.700012)
      Point (X=-229.5, Y=193.700012)
      Point (X=-221.5, Y=193.700012)
      Point (X=-221.5, Y=193.700012)
    Link (From=FM4_ZdvihVytahu, To=M1.0.0, FromPort=EC1, ToPort=EC, IsRoutedByUser=False)
      Point (X=-359.5, Y=367.1)
      Point (X=-359.5, Y=367.1)
      Point (X=-359.5, Y=360.1)
      Point (X=-359.5, Y=280)
      Point (X=-395, Y=280)
      Point (X=-417, Y=280)
      Point (X=-417, Y=280)
    Link (From=FM4_ZdvihVytahu, To=M1.0.0, FromPort=MT1, ToPort=MT, IsRoutedByUser=False)
      Point (X=-331.5, Y=367.1)
      Point (X=-331.5, Y=367.1)
      Point (X=-331.5, Y=360.1)
      Point (X=-331.5, Y=289.3)
      Point (X=-395.4, Y=289.3)
      Point (X=-415.4, Y=289.3)
      Point (X=-415.4, Y=289.3)
    Link (From=FM5_ManipSrobovacky_ZdvihZvarania, To=FM6_ZdvihZakladacaTesnenia, FromPort=PLK2, ToPort=PLK1, IsRoutedByUser=False)
      Point (X=732.1, Y=190.5)
      Point (X=732.1, Y=190.5)
      Point (X=732.1, Y=179.5)
      Point (X=1023.69995, Y=179.5)
      Point (X=1023.69995, Y=172.5)
      Point (X=1031.7, Y=172.5)
      Point (X=1031.7, Y=172.5)
    Link (From=FM5_ManipSrobovacky_ZdvihZvarania, To=M10_ManipSrobovackyOsX, FromPort=EC1, ToPort=EC, IsRoutedByUser=False)
      Point (X=741, Y=317)
      Point (X=741, Y=317)
      Point (X=763, Y=317)
      Point (X=789.5, Y=317)
      Point (X=789.5, Y=379.1)
      Point (X=789.5, Y=386.1)
      Point (X=789.5, Y=386.1)
    Link (From=FM5_ManipSrobovacky_ZdvihZvarania, To=M9_ManipSrobovackyOsY, FromPort=EC2, ToPort=EC, IsRoutedByUser=False)
      Point (X=741, Y=268)
      Point (X=741, Y=268)
      Point (X=763, Y=268)
      Point (X=859.5, Y=268)
      Point (X=859.5, Y=378.1)
      Point (X=859.5, Y=385.1)
      Point (X=859.5, Y=385.1)
    Link (From=FM5_ManipSrobovacky_ZdvihZvarania, To=M6_ZdvihZvaracky, FromPort=EC3, ToPort=EC, IsRoutedByUser=False)
      Point (X=741, Y=219)
      Point (X=741, Y=219)
      Point (X=763, Y=219)
      Point (X=929.5, Y=219)
      Point (X=929.5, Y=378.1)
      Point (X=929.5, Y=385.1)
      Point (X=929.5, Y=385.1)
    Link (From=FM5_ManipSrobovacky_ZdvihZvarania, To=M10_ManipSrobovackyOsX, FromPort=MT1, ToPort=MT, IsRoutedByUser=False)
      Point (X=742.6, Y=326.3)
      Point (X=742.6, Y=326.3)
      Point (X=762.6, Y=326.3)
      Point (X=817.5, Y=326.3)
      Point (X=817.5, Y=379.1)
      Point (X=817.5, Y=386.1)
      Point (X=817.5, Y=386.1)
    Link (From=FM5_ManipSrobovacky_ZdvihZvarania, To=M9_ManipSrobovackyOsY, FromPort=MT2, ToPort=MT, IsRoutedByUser=False)
      Point (X=742.6, Y=277.3)
      Point (X=742.6, Y=277.3)
      Point (X=762.6, Y=277.3)
      Point (X=887.5, Y=277.3)
      Point (X=887.5, Y=378.1)
      Point (X=887.5, Y=385.1)
      Point (X=887.5, Y=385.1)
    Link (From=FM5_ManipSrobovacky_ZdvihZvarania, To=M6_ZdvihZvaracky, FromPort=MT3, ToPort=MT, IsRoutedByUser=False)
      Point (X=742.6, Y=228.3)
      Point (X=742.6, Y=228.3)
      Point (X=762.6, Y=228.3)
      Point (X=957.5, Y=228.3)
      Point (X=957.5, Y=378.1)
      Point (X=957.5, Y=385.1)
      Point (X=957.5, Y=385.1)
    Link (From=FM5_ManipulatorSrobovacky, To=VentilovyTerminal_VT4, FromPort=PLK2, ToPort=PLK1, IsRoutedByUser=False)
      Point (X=-212.9, Y=193.5)
      Point (X=-212.9, Y=193.5)
      Point (X=-212.9, Y=182.5)
      Point (X=-212.9, Y=175)
      Point (X=-196, Y=175)
      Point (X=-196, Y=84.71135)
      Point (X=-196, Y=78.71135)
      Point (X=-196, Y=78.71135)
    Link (From=FM5_ManipulatorSrobovacky, To=M1.1.0, FromPort=EC1, ToPort=EC, IsRoutedByUser=False)
      Point (X=-204, Y=320)
      Point (X=-204, Y=320)
      Point (X=-182, Y=320)
      Point (X=-149.5, Y=320)
      Point (X=-149.5, Y=360.1)
      Point (X=-149.5, Y=367.1)
      Point (X=-149.5, Y=367.1)
    Link (From=FM5_ManipulatorSrobovacky, To=M1.1.1, FromPort=EC2, ToPort=EC, IsRoutedByUser=False)
      Point (X=-204, Y=271)
      Point (X=-204, Y=271)
      Point (X=-182, Y=271)
      Point (X=-66.37523, Y=271)
      Point (X=-66.37523, Y=364.1)
      Point (X=-66.37523, Y=371.1)
      Point (X=-66.37523, Y=371.1)
    Link (From=FM5_ManipulatorSrobovacky, To=M1.1.0, FromPort=MT1, ToPort=MT, IsRoutedByUser=False)
      Point (X=-202.4, Y=329.3)
      Point (X=-202.4, Y=329.3)
      Point (X=-182.4, Y=329.3)
      Point (X=-121.5, Y=329.3)
      Point (X=-121.5, Y=360.1)
      Point (X=-121.5, Y=367.1)
      Point (X=-121.5, Y=367.1)
    Link (From=FM5_ManipulatorSrobovacky, To=M1.1.1, FromPort=MT2, ToPort=MT, IsRoutedByUser=False)
      Point (X=-202.4, Y=280.3)
      Point (X=-202.4, Y=280.3)
      Point (X=-182.4, Y=280.3)
      Point (X=-38.37523, Y=280.3)
      Point (X=-38.37523, Y=364.1)
      Point (X=-38.37523, Y=371.1)
      Point (X=-38.37523, Y=371.1)
    Link (From=FM6_ZdvihZakladacaTesnenia, To=FM7_PojazdZakladacaTesnenia, FromPort=PLK2, ToPort=PLK1, IsRoutedByUser=False)
      Point (X=1040.1, Y=172.5)
      Point (X=1040.1, Y=172.5)
      Point (X=1040.1, Y=161.5)
      Point (X=1040.1, Y=155)
      Point (X=1095, Y=155)
      Point (X=1095, Y=172.5)
      Point (X=1195.7, Y=172.5)
      Point (X=1203.7, Y=172.5)
      Point (X=1203.7, Y=172.5)
    Link (From=FM6_ZdvihZakladacaTesnenia, To=M4_ZdvihZakladacaTesnenia, FromPort=EC1, ToPort=EC, IsRoutedByUser=False)
      Point (X=1049, Y=201)
      Point (X=1049, Y=201)
      Point (X=1071, Y=201)
      Point (X=1105.5, Y=201)
      Point (X=1105.5, Y=378.1)
      Point (X=1105.5, Y=385.1)
      Point (X=1105.5, Y=385.1)
    Link (From=FM6_ZdvihZakladacaTesnenia, To=M4_ZdvihZakladacaTesnenia, FromPort=MT1, ToPort=MT, IsRoutedByUser=False)
      Point (X=1050.6, Y=210.3)
      Point (X=1050.6, Y=210.3)
      Point (X=1070.6, Y=210.3)
      Point (X=1133.5, Y=210.3)
      Point (X=1133.5, Y=378.1)
      Point (X=1133.5, Y=385.1)
      Point (X=1133.5, Y=385.1)
    Link (From=FM7_PojazdZakladacaTesnenia, To=VentilovyTerminal_VT1, FromPort=PLK2, ToPort=PLK1, IsRoutedByUser=False)
      Point (X=1212.1, Y=172.5)
      Point (X=1212.1, Y=180.375)
      Point (X=1195.1, Y=180.375)
      Point (X=1089, Y=180.375)
      Point (X=1089, Y=134)
      Point (X=1082, Y=134)
      Point (X=1082, Y=51)
      Point (X=1082, Y=44)
      Point (X=1082, Y=44)
    Link (From=FM7_PojazdZakladacaTesnenia, To=M5_PojazdZakladacaTesnenia, FromPort=EC1, ToPort=EC, IsRoutedByUser=False)
      Point (X=1221, Y=201)
      Point (X=1221, Y=201)
      Point (X=1243, Y=201)
      Point (X=1286.5, Y=201)
      Point (X=1286.5, Y=378.1)
      Point (X=1286.5, Y=385.1)
      Point (X=1286.5, Y=385.1)
    Link (From=FM7_PojazdZakladacaTesnenia, To=M5_PojazdZakladacaTesnenia, FromPort=MT1, ToPort=MT, IsRoutedByUser=False)
      Point (X=1222.6, Y=210.3)
      Point (X=1222.6, Y=210.3)
      Point (X=1242.6, Y=210.3)
      Point (X=1314.5, Y=210.3)
      Point (X=1314.5, Y=378.1)
      Point (X=1314.5, Y=385.1)
      Point (X=1314.5, Y=385.1)
    Link (From=M4.0.0, To=SD4.0, FromPort=EC, ToPort=EC1, IsRoutedByUser=False)
      Point (X=3312.46167, Y=385.1)
      Point (X=3312.46167, Y=385.1)
      Point (X=3312.46167, Y=378.1)
      Point (X=3312.46167, Y=298)
      Point (X=3277.96167, Y=298)
      Point (X=3255.96167, Y=298)
      Point (X=3255.96167, Y=298)
    Link (From=M4.0.0, To=SD4.0, FromPort=MT, ToPort=MT1, IsRoutedByUser=False)
      Point (X=3340.46167, Y=385.1)
      Point (X=3340.46167, Y=385.1)
      Point (X=3340.46167, Y=378.1)
      Point (X=3340.46167, Y=307.3)
      Point (X=3277.56177, Y=307.3)
      Point (X=3257.56177, Y=307.3)
      Point (X=3257.56177, Y=307.3)
    Link (From=M4.1.0, To=SD4.1, FromPort=EC, ToPort=EC1, IsRoutedByUser=False)
      Point (X=3473.46167, Y=385.1)
      Point (X=3473.46167, Y=385.1)
      Point (X=3473.46167, Y=378.1)
      Point (X=3473.46167, Y=298)
      Point (X=3437.96167, Y=298)
      Point (X=3415.96167, Y=298)
      Point (X=3415.96167, Y=298)
    Link (From=M4.1.0, To=SD4.1, FromPort=MT, ToPort=MT1, IsRoutedByUser=False)
      Point (X=3501.46167, Y=385.1)
      Point (X=3501.46167, Y=385.1)
      Point (X=3501.46167, Y=378.1)
      Point (X=3501.46167, Y=307.3)
      Point (X=3437.56177, Y=307.3)
      Point (X=3417.56177, Y=307.3)
      Point (X=3417.56177, Y=307.3)
    Link (From=P1_CAM3, To=RJ7_P1_Srobovacka_M4, FromPort=PN1, ToPort=PN2, IsRoutedByUser=False)
      Point (X=46, Y=467)
      Point (X=46, Y=467)
      Point (X=46, Y=479)
      Point (X=46, Y=485)
      Point (X=234.30896, Y=485)
      Point (X=234.30896, Y=273)
      Point (X=234.30896, Y=261)
      Point (X=234.30896, Y=261)
    Link (From=P1_CAM3, To=R2_IRB1200, FromPort=PN2, ToPort=PN1, IsRoutedByUser=True)
      Point (X=1476, Y=546)
      Point (X=1476, Y=546)
      Point (X=1456, Y=546)
      Point (X=1445, Y=546)
      Point (X=1445, Y=483.558136)
      Point (X=249.30896, Y=483.558136)
      Point (X=249.30896, Y=273)
      Point (X=249.30896, Y=261)
      Point (X=249.30896, Y=261)
    Link (From=P3_Srobovacka_K40, To=RJ1_P2_SrobovackaMatic_M4, FromPort=PN1, ToPort=PN2, IsRoutedByUser=True)
      Point (X=2266, Y=467)
      Point (X=2266, Y=467)
      Point (X=2246, Y=467)
      Point (X=2085, Y=467)
      Point (X=2085, Y=625)
      Point (X=2055, Y=625)
      Point (X=2055, Y=1085)
      Point (X=1492, Y=1085)
      Point (X=1492, Y=1078)
      Point (X=1492, Y=1066)
      Point (X=1492, Y=1066)
    Link (From=P3_Srobovacka_K40, To=P3_Srobovacka_M5, FromPort=PN2, ToPort=PN1, IsRoutedByUser=False)
      Point (X=2281, Y=467)
      Point (X=2281, Y=467)
      Point (X=2281, Y=479)
      Point (X=2281, Y=485)
      Point (X=2347, Y=485)
      Point (X=2347, Y=467)
      Point (X=2392, Y=467)
      Point (X=2412, Y=467)
      Point (X=2412, Y=467)
    Link (From=PS1.1, To=SI1.2, FromPort=X2X1, ToPort=X2X2, IsRoutedByUser=True)
      Point (X=-424, Y=1061)
      Point (X=-424, Y=1061)
      Point (X=-435, Y=1061)
      Point (X=-445, Y=1061)
      Point (X=-445, Y=1036.10327)
      Point (X=204.046982, Y=1036.10327)
      Point (X=204.046982, Y=537)
      Point (X=200, Y=537)
      Point (X=188, Y=537)
      Point (X=188, Y=537)
    Link (From=PS4.1, To=SI4.2, FromPort=X2X1, ToPort=X2X2, IsRoutedByUser=False)
      Point (X=3553.96167, Y=535)
      Point (X=3553.96167, Y=535)
      Point (X=3565.96167, Y=535)
      Point (X=3585.96167, Y=535)
      Point (X=3596.96167, Y=535)
      Point (X=3596.96167, Y=535)
    Link (From=R1_IRB120, To=RJ5_P1_Srobovacka_K30, FromPort=PN2, ToPort=PN1, IsRoutedByUser=True)
      Point (X=31, Y=266)
      Point (X=31, Y=266)
      Point (X=31, Y=278)
      Point (X=31, Y=285)
      Point (X=-12.1752958, Y=285)
      Point (X=-12.1752958, Y=171.462219)
      Point (X=46, Y=171.462219)
      Point (X=46, Y=87)
      Point (X=46, Y=75)
      Point (X=46, Y=75)
    Link (From=R2_IRB1200, To=RJ2_P2_Srobovacka_M6, FromPort=PN2, ToPort=PN1, IsRoutedByUser=False)
      Point (X=1492.46167, Y=546)
      Point (X=1492.46167, Y=546)
      Point (X=1492.46167, Y=558)
      Point (X=1492.46167, Y=571)
      Point (X=1446.93164, Y=571)
      Point (X=1446.93164, Y=711)
      Point (X=1477.46167, Y=711)
      Point (X=1477.46167, Y=698)
      Point (X=1477.46167, Y=686)
      Point (X=1477.46167, Y=686)
    Link (From=RJ1_P2_SrobovackaMatic_M4, To=RJ3_P2_Srobovacka_M4, FromPort=PN1, ToPort=PN2, IsRoutedByUser=False)
      Point (X=1491, Y=970)
      Point (X=1491, Y=970)
      Point (X=1491, Y=982)
      Point (X=1491, Y=1002)
      Point (X=1451, Y=1002)
      Point (X=1451, Y=1085)
      Point (X=1477.46167, Y=1085)
      Point (X=1477.46167, Y=1078)
      Point (X=1477.46167, Y=1066)
      Point (X=1477.46167, Y=1066)
    Link (From=RJ2_P2_Srobovacka_M6, To=RJ4_P2_Srobovacka_M5, FromPort=PN2, ToPort=PN1, IsRoutedByUser=False)
      Point (X=1492.46167, Y=686)
      Point (X=1492.46167, Y=686)
      Point (X=1492.46167, Y=698)
      Point (X=1492.46167, Y=718)
      Point (X=1446.93164, Y=718)
      Point (X=1446.93164, Y=844)
      Point (X=1477.46167, Y=844)
      Point (X=1477.46167, Y=838)
      Point (X=1477.46167, Y=826)
      Point (X=1477.46167, Y=826)
    Link (From=RJ3_P2_Srobovacka_M4, To=RJ4_P2_Srobovacka_M5, FromPort=PN1, ToPort=PN2, IsRoutedByUser=True)
      Point (X=1476.93164, Y=970)
      Point (X=1476.93164, Y=970)
      Point (X=1476.93164, Y=982)
      Point (X=1476.93164, Y=991)
      Point (X=1447.93164, Y=991)
      Point (X=1447.93164, Y=878)
      Point (X=1491.93164, Y=878)
      Point (X=1491.93164, Y=838)
      Point (X=1491.93164, Y=826)
      Point (X=1491.93164, Y=826)
    Link (From=RJ5_P1_Srobovacka_K30, To=RJ6_P1_Srobovacka_M5, FromPort=PN2, ToPort=PN1, IsRoutedByUser=False)
      Point (X=46.6299133, Y=266)
      Point (X=46.6299133, Y=266)
      Point (X=46.6299133, Y=278)
      Point (X=46.6299133, Y=295)
      Point (X=-5, Y=295)
      Point (X=-5, Y=388)
      Point (X=27.3078, Y=388)
      Point (X=27.3078, Y=380)
      Point (X=27.3078, Y=368)
      Point (X=27.3078, Y=368)
    Link (From=RJ6_P1_Srobovacka_M5, To=RJ7_P1_Srobovacka_M4, FromPort=PN2, ToPort=PN1, IsRoutedByUser=False)
      Point (X=46.6299133, Y=368)
      Point (X=46.6299133, Y=368)
      Point (X=46.6299133, Y=380)
      Point (X=46.6299133, Y=395)
      Point (X=5, Y=395)
      Point (X=5, Y=488)
      Point (X=31.6299133, Y=488)
      Point (X=31.6299133, Y=479)
      Point (X=31.6299133, Y=467)
      Point (X=31.6299133, Y=467)
    Link (From=SI2.1, To=SI2.2, FromPort=X2X2, ToPort=X2X1, IsRoutedByUser=False)
      Point (X=857.980469, Y=537)
      Point (X=857.980469, Y=537)
      Point (X=869.980469, Y=537)
      Point (X=880, Y=537)
      Point (X=891, Y=537)
      Point (X=891, Y=537)
    Link (From=SI4.1, To=X67DI1371.L08j, FromPort=X2X1, ToPort=X2X2, IsRoutedByUser=False)
      Point (X=3403.96167, Y=535)
      Point (X=3403.96167, Y=535)
      Point (X=3415.96167, Y=535)
      Point (X=3435.96167, Y=535)
      Point (X=3446.96167, Y=535)
      Point (X=3446.96167, Y=535)
    Link (From=SI4.1, To=SI4.2, FromPort=X2X2, ToPort=X2X1, IsRoutedByUser=False)
      Point (X=3478.96167, Y=535)
      Point (X=3478.96167, Y=535)
      Point (X=3490.96167, Y=535)
      Point (X=3510.96167, Y=535)
      Point (X=3521.96167, Y=535)
      Point (X=3521.96167, Y=535)
    Link (From=VentilovyTerminal_VT1, To=VentilovyTerminal_VT2, FromPort=PLK2, ToPort=PLK1, IsRoutedByUser=False)
      Point (X=1107, Y=44)
      Point (X=1107, Y=44)
      Point (X=1107, Y=51)
      Point (X=1107, Y=65)
      Point (X=1190, Y=65)
      Point (X=1190, Y=51)
      Point (X=1190, Y=44)
      Point (X=1190, Y=44)
    Link (From=VentilovyTerminal_VT2, To=VentilovyTerminal_VT3, FromPort=PLK2, ToPort=PLK1, IsRoutedByUser=False)
      Point (X=1215, Y=44)
      Point (X=1215, Y=44)
      Point (X=1215, Y=51)
      Point (X=1215, Y=65)
      Point (X=1298, Y=65)
      Point (X=1298, Y=51)
      Point (X=1298, Y=44)
      Point (X=1298, Y=44)
    Link (From=VentilovyTerminal_VT4, To=VentilovyTerminal_VT5, FromPort=PLK2, ToPort=PLK1, IsRoutedByUser=False)
      Point (X=-171, Y=78.71135)
      Point (X=-171, Y=78.71135)
      Point (X=-171, Y=84.71135)
      Point (X=-171, Y=95)
      Point (X=-85, Y=95)
      Point (X=-85, Y=84.71135)
      Point (X=-85, Y=78.71135)
      Point (X=-85, Y=78.71135)
    Link (From=VentilovyTerminal_VT6, To=VentilovyTerminal_VT7, FromPort=PLK2, ToPort=PLK1, IsRoutedByUser=False)
      Point (X=2253.644, Y=248)
      Point (X=2253.644, Y=248)
      Point (X=2253.644, Y=255)
      Point (X=2253.644, Y=265)
      Point (X=2363, Y=265)
      Point (X=2363, Y=255)
      Point (X=2363, Y=248)
      Point (X=2363, Y=248)
    Link (From=X67DI1371.L08j, To=X67DI1371a, FromPort=X2X1, ToPort=X2X2, IsRoutedByUser=False)
      Point (X=3328.96167, Y=535)
      Point (X=3328.96167, Y=535)
      Point (X=3340.96167, Y=535)
      Point (X=3360.96167, Y=535)
      Point (X=3371.96167, Y=535)
      Point (X=3371.96167, Y=535)
  InfoElements:
    InfoElementText (Id=Textbox_3, X=-680.0337, Y=-360, Width=1216, Height=1945.42822)
      Text = Bunka č.1 (Color=Black, FontName=Arial, FontSize=20, FontStyle=Regular, AlignmentHorizontal=Center)
      Background (Color=White, Transparent=False)
      Border (Color=Black, Transparent=False, DashStyle=Solid, Width=1)
    InfoElementText (Id=Textbox_5, X=1983.96631, Y=-360, Width=723.1748, Height=1873.79407)
      Text = Bunka č.3 (Color=Black, FontName=Arial, FontSize=20, FontStyle=Regular, AlignmentHorizontal=Center)
      Background (Color=White, Transparent=False)
      Border (Color=Black, Transparent=False, DashStyle=Solid, Width=1)
    InfoElementText (Id=Textbox_6, X=3201.96167, Y=-362, Width=723.1748, Height=1873.79407)
      Text = Bunka č.4 (Color=Black, FontName=Arial, FontSize=20, FontStyle=Regular, AlignmentHorizontal=Center)
      Background (Color=White, Transparent=False)
      Border (Color=Black, Transparent=False, DashStyle=Solid, Width=1)
    InfoElementText (Id=Textbox_8, X=2049.41528, Y=-281.439362, Width=146.228638, Height=136.421783)
      Text = ETH/PNT switch (Color=Black, FontName=Arial, FontSize=20, FontStyle=Regular, AlignmentHorizontal=Left)
      Background (Color=White, Transparent=False)
      Border (Color=Black, Transparent=False, DashStyle=Solid, Width=1)
    InfoElementText (Id=Textbox_9, X=2483.96631, Y=-300, Width=141.222534, Height=136.987244)
      Text = PWL hub (Color=Black, FontName=Arial, FontSize=20, FontStyle=Regular, AlignmentHorizontal=Left)
      Background (Color=White, Transparent=False)
      Border (Color=Black, Transparent=False, DashStyle=Solid, Width=1)
    InfoElementText (Id=Textbox_10, X=9.15527344E-05, Y=-281.439331, Width=146.228638, Height=136.421783)
      Text = ETH/ PNT switch (Color=Black, FontName=Arial, FontSize=20, FontStyle=Regular, AlignmentHorizontal=Left)
      Background (Color=White, Transparent=False)
      Border (Color=Black, Transparent=False, DashStyle=Solid, Width=1)
    InfoElementText (Id=Textbox_11, X=1119.70117, Y=-281.4394, Width=146.228638, Height=136.421783)
      Text = ETH/ PNT switch (Color=Black, FontName=Arial, FontSize=20, FontStyle=Regular, AlignmentHorizontal=Left)
      Background (Color=White, Transparent=False)
      Border (Color=Black, Transparent=False, DashStyle=Solid, Width=1)
    InfoElementText (Id=Textbox_12, X=3693.37378, Y=-263.336548, Width=146.228638, Height=136.421783)
      Text = ETH/ PNT switch (Color=Black, FontName=Arial, FontSize=20, FontStyle=Regular, AlignmentHorizontal=Left)
      Background (Color=White, Transparent=False)
      Border (Color=Black, Transparent=False, DashStyle=Solid, Width=1)
    InfoElementText (Id=Textbox_13, X=653.0823, Y=-358.879425, Width=987.4723, Height=1869.125)
      Text = Bunka č.2 (Color=Black, FontName=Arial, FontSize=20, FontStyle=Regular, AlignmentHorizontal=Center)
      Background (Color=White, Transparent=False)
      Border (Color=Black, Transparent=False, DashStyle=Solid, Width=1)
    InfoElementText (Id=Textbox_14, X=768, Y=-302.4394, Width=97, Height=21)
      Text = 192.168.1.21 (Color=Black, FontName=Arial, FontSize=12, FontStyle=Regular, AlignmentHorizontal=Left)
      Background (Color=White, Transparent=False)
      Border (Color=Black, Transparent=False, DashStyle=Solid, Width=1)
    InfoElementText (Id=Textbox_15, X=748, Y=-18, Width=20, Height=18)
      Text = 21 (Color=Black, FontName=Arial, FontSize=12, FontStyle=Regular, AlignmentHorizontal=Left)
      Background (Color=White, Transparent=False)
      Border (Color=Black, Transparent=False, DashStyle=Solid, Width=1)
    InfoElementText (Id=Textbox_16, X=1191, Y=-18, Width=20, Height=18)
      Text = 26 (Color=Black, FontName=Arial, FontSize=12, FontStyle=Regular, AlignmentHorizontal=Left)
      Background (Color=White, Transparent=False)
      Border (Color=Black, Transparent=False, DashStyle=Solid, Width=1)
    InfoElementText (Id=Textbox_17, X=1077, Y=-18, Width=20, Height=18)
      Text = 25 (Color=Black, FontName=Arial, FontSize=12, FontStyle=Regular, AlignmentHorizontal=Left)
      Background (Color=White, Transparent=False)
      Border (Color=Black, Transparent=False, DashStyle=Solid, Width=1)
    InfoElementText (Id=Textbox_18, X=1302, Y=-18, Width=20, Height=18)
      Text = 27 (Color=Black, FontName=Arial, FontSize=12, FontStyle=Regular, AlignmentHorizontal=Left)
      Background (Color=White, Transparent=False)
      Border (Color=Black, Transparent=False, DashStyle=Solid, Width=1)
    InfoElementText (Id=Textbox_19, X=1049, Y=133, Width=20, Height=18)
      Text = 23 (Color=Black, FontName=Arial, FontSize=12, FontStyle=Regular, AlignmentHorizontal=Left)
      Background (Color=White, Transparent=False)
      Border (Color=Black, Transparent=False, DashStyle=Solid, Width=1)
    InfoElementText (Id=Textbox_20, X=1211, Y=144, Width=20, Height=18)
      Text = 24 (Color=Black, FontName=Arial, FontSize=12, FontStyle=Regular, AlignmentHorizontal=Left)
      Background (Color=White, Transparent=False)
      Border (Color=Black, Transparent=False, DashStyle=Solid, Width=1)
    InfoElementText (Id=Textbox_21, X=700, Y=151, Width=20, Height=18)
      Text = 22 (Color=Black, FontName=Arial, FontSize=12, FontStyle=Regular, AlignmentHorizontal=Left)
      Background (Color=White, Transparent=False)
      Border (Color=Black, Transparent=False, DashStyle=Solid, Width=1)
    InfoElementText (Id=Textbox_22, X=2257.46631, Y=34.7113457, Width=20, Height=15.2886543)
      Text = 2 (Color=Black, FontName=Arial, FontSize=12, FontStyle=Regular, AlignmentHorizontal=Left)
      Background (Color=White, Transparent=False)
      Border (Color=Black, Transparent=False, DashStyle=Solid, Width=1)
    InfoElementText (Id=Textbox_23, X=2280.96631, Y=-110.7, Width=97, Height=21)
      Text = 192.168.1.1 (Color=Black, FontName=Arial, FontSize=12, FontStyle=Regular, AlignmentHorizontal=Left)
      Background (Color=White, Transparent=False)
      Border (Color=Black, Transparent=False, DashStyle=Solid, Width=1)
    InfoElementText (Id=Textbox_24, X=-338, Y=-323.4394, Width=97, Height=21)
      Text = 192.168.1.11 (Color=Black, FontName=Arial, FontSize=12, FontStyle=Regular, AlignmentHorizontal=Left)
      Background (Color=White, Transparent=False)
      Border (Color=Black, Transparent=False, DashStyle=Solid, Width=1)
    InfoElementText (Id=Textbox_25, X=-408, Y=-10, Width=20, Height=18)
      Text = 11 (Color=Black, FontName=Arial, FontSize=12, FontStyle=Regular, AlignmentHorizontal=Left)
      Background (Color=White, Transparent=False)
      Border (Color=Black, Transparent=False, DashStyle=Solid, Width=1)
    InfoElementText (Id=Textbox_26, X=-388, Y=241, Width=20, Height=18)
      Text = 12 (Color=Black, FontName=Arial, FontSize=12, FontStyle=Regular, AlignmentHorizontal=Left)
      Background (Color=White, Transparent=False)
      Border (Color=Black, Transparent=False, DashStyle=Solid, Width=1)
    InfoElementText (Id=Textbox_27, X=-207, Y=151, Width=22, Height=18)
      Text = 13 (Color=Black, FontName=Arial, FontSize=12, FontStyle=Regular, AlignmentHorizontal=Left)
      Background (Color=White, Transparent=False)
      Border (Color=Black, Transparent=False, DashStyle=Solid, Width=1)
    InfoElementText (Id=Textbox_28, X=-192.875229, Y=8.711346, Width=22.8752289, Height=23.1730957)
      Text = 14 (Color=Black, FontName=Arial, FontSize=12, FontStyle=Regular, AlignmentHorizontal=Left)
      Background (Color=White, Transparent=False)
      Border (Color=Black, Transparent=False, DashStyle=Solid, Width=1)
    InfoElementText (Id=Textbox_30, X=-87.87523, Y=8.711346, Width=22.8752289, Height=23.1730957)
      Text = 15 (Color=Black, FontName=Arial, FontSize=12, FontStyle=Regular, AlignmentHorizontal=Left)
      Background (Color=White, Transparent=False)
      Border (Color=Black, Transparent=False, DashStyle=Solid, Width=1)
    InfoElementText (Id=Textbox_32, X=8.3078, Y=13.7113457, Width=106.629913, Height=21)
      Text = 192.168.1.101 (Color=Black, FontName=Arial, FontSize=12, FontStyle=Regular, AlignmentHorizontal=Left)
      Background (Color=White, Transparent=False)
      Border (Color=Black, Transparent=False, DashStyle=Solid, Width=1)
    InfoElementText (Id=Textbox_33, X=1458.46167, Y=486, Width=106.629913, Height=21)
      Text = 192.168.1.102 (Color=Black, FontName=Arial, FontSize=12, FontStyle=Regular, AlignmentHorizontal=Left)
      Background (Color=White, Transparent=False)
      Border (Color=Black, Transparent=False, DashStyle=Solid, Width=1)
    InfoElementText (Id=Textbox_34, X=8.3078, Y=204, Width=106.629913, Height=21)
      Text = 192.168.1.103 (Color=Black, FontName=Arial, FontSize=12, FontStyle=Regular, AlignmentHorizontal=Left)
      Background (Color=White, Transparent=False)
      Border (Color=Black, Transparent=False, DashStyle=Solid, Width=1)
    InfoElementText (Id=Textbox_35, X=8.3078, Y=308, Width=106.629913, Height=21)
      Text = 192.168.1.104 (Color=Black, FontName=Arial, FontSize=12, FontStyle=Regular, AlignmentHorizontal=Left)
      Background (Color=White, Transparent=False)
      Border (Color=Black, Transparent=False, DashStyle=Solid, Width=1)
    InfoElementText (Id=Textbox_36, X=12.6299133, Y=407, Width=106.629913, Height=21)
      Text = 192.168.1.105 (Color=Black, FontName=Arial, FontSize=12, FontStyle=Regular, AlignmentHorizontal=Left)
      Background (Color=White, Transparent=False)
      Border (Color=Black, Transparent=False, DashStyle=Solid, Width=1)
    InfoElementText (Id=Textbox_37, X=2049.41528, Y=2, Width=20, Height=18)
      Text = 31 (Color=Black, FontName=Arial, FontSize=12, FontStyle=Regular, AlignmentHorizontal=Left)
      Background (Color=White, Transparent=False)
      Border (Color=Black, Transparent=False, DashStyle=Solid, Width=1)
    InfoElementText (Id=Textbox_38, X=2080.2, Y=204, Width=24, Height=18)
      Text = 32 (Color=Black, FontName=Arial, FontSize=12, FontStyle=Regular, AlignmentHorizontal=Left)
      Background (Color=White, Transparent=False)
      Border (Color=Black, Transparent=False, DashStyle=Solid, Width=1)
    InfoElementText (Id=Textbox_39, X=1458.46167, Y=626, Width=106.629913, Height=21)
      Text = 192.168.1.106 (Color=Black, FontName=Arial, FontSize=12, FontStyle=Regular, AlignmentHorizontal=Left)
      Background (Color=White, Transparent=False)
      Border (Color=Black, Transparent=False, DashStyle=Solid, Width=1)
    InfoElementText (Id=Textbox_40, X=1458.46167, Y=764, Width=106.629913, Height=21)
      Text = 192.168.1.107 (Color=Black, FontName=Arial, FontSize=12, FontStyle=Regular, AlignmentHorizontal=Left)
      Background (Color=White, Transparent=False)
      Border (Color=Black, Transparent=False, DashStyle=Solid, Width=1)
    InfoElementText (Id=Textbox_41, X=1458.46167, Y=910, Width=106.629913, Height=21)
      Text = 192.168.1.108 (Color=Black, FontName=Arial, FontSize=12, FontStyle=Regular, AlignmentHorizontal=Left)
      Background (Color=White, Transparent=False)
      Border (Color=Black, Transparent=False, DashStyle=Solid, Width=1)
    InfoElementText (Id=Textbox_42, X=2223, Y=186, Width=24, Height=18)
      Text = 33 (Color=Black, FontName=Arial, FontSize=12, FontStyle=Regular, AlignmentHorizontal=Left)
      Background (Color=White, Transparent=False)
      Border (Color=Black, Transparent=False, DashStyle=Solid, Width=1)
    InfoElementText (Id=Textbox_43, X=2355, Y=185, Width=24, Height=19)
      Text = 34 (Color=Black, FontName=Arial, FontSize=12, FontStyle=Regular, AlignmentHorizontal=Left)
      Background (Color=White, Transparent=False)
      Border (Color=Black, Transparent=False, DashStyle=Solid, Width=1)
    InfoElementText (Id=Textbox_45, X=2236.37, Y=407, Width=106.629913, Height=21)
      Text = 192.168.1.110 (Color=Black, FontName=Arial, FontSize=12, FontStyle=Regular, AlignmentHorizontal=Left)
      Background (Color=White, Transparent=False)
      Border (Color=Black, Transparent=False, DashStyle=Solid, Width=1)
    InfoElementText (Id=Textbox_46, X=2393, Y=407, Width=106.629913, Height=21)
      Text = 192.168.1.111 (Color=Black, FontName=Arial, FontSize=12, FontStyle=Regular, AlignmentHorizontal=Left)
      Background (Color=White, Transparent=False)
      Border (Color=Black, Transparent=False, DashStyle=Solid, Width=1)
    InfoElementText (Id=Textbox_47, X=1458.46167, Y=1006, Width=106.629913, Height=21)
      Text = 192.168.1.109 (Color=Black, FontName=Arial, FontSize=12, FontStyle=Regular, AlignmentHorizontal=Left)
      Background (Color=White, Transparent=False)
      Border (Color=Black, Transparent=False, DashStyle=Solid, Width=1)
    InfoElementText (Id=Textbox_48, X=198.679047, Y=201, Width=106.629913, Height=21)
      Text = 192.168.1.121 (Color=Black, FontName=Arial, FontSize=12, FontStyle=Regular, AlignmentHorizontal=Left)
      Background (Color=White, Transparent=False)
      Border (Color=Black, Transparent=False, DashStyle=Solid, Width=1)
```
